// TIA Portal V20 export
TYPE "LBP_typePowerrideConfigPos"
TITLE = Data type for configuration of a Powerride position / Type de données pour configuration d'une position Powerride
// User data type for LBP_PowerrideConfig (sub type) / Type de données utilisateur pour LBP_PowerrideConfig (sous-type)
   STRUCT
      value { S7_SetPoint := 'True'} : USInt;   // override factor / facteur de correction
      ledColor { S7_SetPoint := 'True'} : USInt;   // color of scale LEDs / couleur des LED d'échelle
      vibrationIndex { S7_SetPoint := 'True'} : USInt;   // index of vibration pattern / indice du modèle de vibration
   END_STRUCT;
END_TYPE
